// TIA Portal project "Es03_SCHELETRO" (V18)

(* hardware
DEVICE "S71500/ET200MP station_1"  S7-1500 station
   slot 0: "Telaio di montaggio_0"  Rack  6ES7 590-1***0-0AA0
   slot 1: "PLC_1"  CPU 1516-3 PN/DP  6ES7 516-3AN01-0AB0  V2.5
      slot 3: "Display CPU_1"  6ES7591-1BA00-0AA0
   slot 2: "DI 32x24VDC HF_1"  DI 32x24VDC HF  6ES7 521-1BL00-0AB0  V2.1
   slot 3: "DQ 32x24VDC/0.5A HF_1"  DQ 32x24VDC/0.5A HF  6ES7 522-1BL01-0AB0  V1.0
   slot 4: "AI 8xU/I/RTD/TC ST_1"  AI 8xU/I/RTD/TC ST  6ES7 531-7KF00-0AB0  V2.1
   slot 5: "AQ 4xU/I ST_1"  AQ 4xU/I ST  6ES7 532-5HD00-0AB0  V2.1
*)

// ===== PLC "PLC_1"  CPU 1516-3 PN/DP =====

DATA_BLOCK "DB_Comandi"   // DB1
{ S7_Optimized_Access := 'TRUE' }
VERSION : 0.1
   VAR
      btnStop : Bool;
      btnAuto : Bool;
      btnMan : Bool;
      btnReset : Bool;
      btnEmergenza : Bool;
   END_VAR
BEGIN
END_DATA_BLOCK

DATA_BLOCK "DB_Stati"   // DB2
{ S7_Optimized_Access := 'TRUE' }
VERSION : 0.1
   VAR
      sAuto : Bool;
      sStop : Bool;
      sMan : Bool;
      sHome : Bool;
      sAttesaStop : Bool;
      sEmergenza : Bool;
      blni1 : Bool;
      blni2 : Bool;
      bRip1 : Bool;
      bRip2 : Bool;
   END_VAR
BEGIN
END_DATA_BLOCK

DATA_BLOCK "DB_Tappe"   // DB3
{ S7_Optimized_Access := 'TRUE' }
VERSION : 0.1
   VAR
      tappeGemma : Int;
      tappeM1 : Int;
      tappeM2 : Int;
   END_VAR
BEGIN
END_DATA_BLOCK

DATA_BLOCK "DB_Variabili"   // DB4
{ S7_Optimized_Access := 'TRUE' }
VERSION : 0.1
   VAR
      timerResetPulsantiSTART : Bool;
      timerResetPulsantiDONE : Bool;
      timerResetPulsantiOUTPUT : Time;
      timerResetPulsantiDURATA : Time;
   END_VAR
BEGIN
END_DATA_BLOCK

// folder: System blocks/Program resources

DATA_BLOCK "timerResetPulsanti"   // DB5
{ S7_Optimized_Access := 'TRUE' }
AUTHOR : Simatic
FAMILY : IEC
NAME : IEC_TMR
VERSION : 1.0
// stored: InstanceOfName IEC_TIMER
"IEC_TIMER"
BEGIN
END_DATA_BLOCK

// folder: (top level)

FUNCTION "FC_Gemma" : Void   // FC1, SCL
{ S7_Optimized_Access := 'TRUE' }
VERSION : 0.1
BEGIN
   CASE "DB_Tappe".tappeGemma OF
       0: //Stato di Riposo
           "DB_Stati".sStop := TRUE;
           IF "DB_Comandi".btnAuto = TRUE THEN
               "DB_Tappe".tappeGemma := 1; //Home
               "DB_Stati".sAttesaStop := FALSE;
               "DB_Stati".sAuto := FALSE;
               "DB_Stati".sHome := TRUE;
               "DB_Stati".sMan := FALSE;
               "DB_Stati".sStop := FALSE;
               "DB_Stati".sEmergenza := FALSE;
           ELSE
               IF "DB_Comandi".btnMan = TRUE THEN
                   "DB_Tappe".tappeGemma := 4; //Manuale
                   "DB_Stati".sAttesaStop := FALSE;
                   "DB_Stati".sAuto := FALSE;
                   "DB_Stati".sHome := FALSE;
                   "DB_Stati".sMan := TRUE;
                   "DB_Stati".sStop := FALSE;
                   "DB_Stati".sEmergenza := FALSE;
               END_IF;
           END_IF;

        1: //Stato di Home
            IF "DB_Stati".blni1 = TRUE AND "DB_Stati".blni2 = TRUE THEN
                "DB_Tappe".tappeGemma := 2; //Automatico
                "DB_Stati".sAttesaStop := FALSE;
                "DB_Stati".sAuto := TRUE;
                "DB_Stati".sHome := FALSE;
                "DB_Stati".sMan := FALSE;
                "DB_Stati".sStop := FALSE;
                "DB_Stati".sEmergenza := FALSE;
            END_IF;

        2: //Stato di Automatico
            IF "DB_Comandi".btnStop = TRUE THEN
                "DB_Tappe".tappeGemma := 3; //Attesa Stop
                "DB_Stati".sAttesaStop := TRUE;
                "DB_Stati".sAuto := FALSE;
                "DB_Stati".sHome := FALSE;
                "DB_Stati".sMan := FALSE;
                "DB_Stati".sStop := FALSE;
                "DB_Stati".sEmergenza := FALSE;
            END_IF;

        3: //Stato di Attesa Stop
            IF "DB_Stati".bRip1 = TRUE AND "DB_Stati".bRip2 = TRUE THEN
                "DB_Tappe".tappeGemma := 0; //Stop
                "DB_Stati".sAttesaStop := FALSE;
                "DB_Stati".sAuto := FALSE;
                "DB_Stati".sHome := FALSE;
                "DB_Stati".sMan := FALSE;
                "DB_Stati".sStop := TRUE;
                "DB_Stati".sEmergenza := FALSE;
            END_IF;

        4: //Stato di Manuale
            IF "DB_Comandi".btnStop = TRUE THEN
                "DB_Tappe".tappeGemma := 0; //Stop
                "DB_Stati".sAttesaStop := FALSE;
                "DB_Stati".sAuto := FALSE;
                "DB_Stati".sHome := FALSE;
                "DB_Stati".sMan := FALSE;
                "DB_Stati".sStop := TRUE;
                "DB_Stati".sEmergenza := FALSE;
            END_IF;

        5: //Stato di Emergenza
            IF "DB_Comandi".btnEmergenza = TRUE AND "DB_Stati".sEmergenza THEN
                "DB_Tappe".tappeGemma := 0; //Stop
                "DB_Stati".sAttesaStop := FALSE;
                "DB_Stati".sAuto := FALSE;
                "DB_Stati".sHome := FALSE;
                "DB_Stati".sMan := FALSE;
                "DB_Stati".sStop := TRUE;
                "DB_Stati".sEmergenza := FALSE;
            END_IF;
    END_CASE;

    //Gestione Emergenza
    //
    IF "DB_Comandi".btnEmergenza = FALSE THEN
        "DB_Tappe".tappeGemma := 5; //Emergenza
        "DB_Stati".sAttesaStop := FALSE;
        "DB_Stati".sAuto := FALSE;
        "DB_Stati".sHome := FALSE;
        "DB_Stati".sMan := FALSE;
        "DB_Stati".sStop := FALSE;
        "DB_Stati".sEmergenza := TRUE;
    END_IF;
END_FUNCTION

FUNCTION "FC_Grafset" : Void   // FC2, SCL
{ S7_Optimized_Access := 'TRUE' }
VERSION : 0.1
BEGIN
   //Imposto bIni e bRip a TRUE. Andranno poi gestiti in base alle condizioni dell'impianto
   //
   "DB_Stati".blni1 := TRUE;
   "DB_Stati".blni2 := TRUE;
   "DB_Stati".bRip1 := TRUE;
   "DB_Stati".bRip2 := TRUE;
END_FUNCTION

FUNCTION "FC_ResetPulsanti" : Void   // FC3, SCL
{ S7_Optimized_Access := 'TRUE' }
VERSION : 0.1
BEGIN
   IF "DB_Comandi".btnAuto = TRUE OR
       "DB_Comandi".btnMan = TRUE OR
       "DB_Comandi".btnReset = TRUE OR
       "DB_Comandi".btnStop = TRUE THEN
       "DB_Variabili".timerResetPulsantiSTART := TRUE;
   END_IF;

   IF "DB_Variabili".timerResetPulsantiDONE = TRUE THEN
       "DB_Variabili".timerResetPulsantiSTART := FALSE;
       "DB_Variabili".timerResetPulsantiDONE := FALSE;
       "DB_Comandi".btnAuto := FALSE;
       "DB_Comandi".btnMan := FALSE;
       "DB_Comandi".btnReset := FALSE;
       "DB_Comandi".btnStop := FALSE;
   END_IF;
END_FUNCTION

FUNCTION "FC_Timer" : Void   // FC4, SCL
{ S7_Optimized_Access := 'TRUE' }
VERSION : 0.1
BEGIN
   "DB_Variabili".timerResetPulsantiDURATA := T#500ms;

   "timerResetPulsanti".TON(IN:="DB_Variabili".timerResetPulsantiSTART,
                            PT:="DB_Variabili".timerResetPulsantiDURATA,
                            Q=>"DB_Variabili".timerResetPulsantiDONE,
                            ET=>"DB_Variabili".timerResetPulsantiOUTPUT);
END_FUNCTION

FUNCTION "FC_Uscite" : Void   // FC5, SCL
{ S7_Optimized_Access := 'TRUE' }
VERSION : 0.1
BEGIN
END_FUNCTION

ORGANIZATION_BLOCK "Main"   // OB1, LAD, ProgramCycle
TITLE = "Main Program Sweep (Cycle)"
{ S7_Optimized_Access := 'TRUE' }
VERSION : 0.1
   VAR_INPUT
      Initial_Call : Bool;   // Initial call of this OB
      Remanence : Bool;   // =True, if remanent data are available
   END_VAR
   VAR_TEMP   // added for the SCL form of the ladder/FBD networks
      _w1 : Bool;
      _w2 : Bool;
      _w3 : Bool;
      _w4 : Bool;
   END_VAR
BEGIN

REGION Network 1
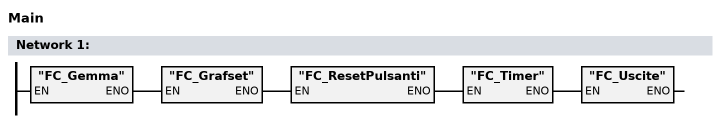
   RUNG wire#powerrail
      "FC_Gemma"()
      "FC_Grafset"()
      "FC_ResetPulsanti"()
      "FC_Timer"()
      "FC_Uscite"()
   END_RUNG
   // the same network as SCL:
   "FC_Gemma"(ENO => #_w1);
   "FC_Grafset"(EN := #_w1, ENO => #_w2);
   "FC_ResetPulsanti"(EN := #_w2, ENO => #_w3);
   "FC_Timer"(EN := #_w3, ENO => #_w4);
   IF #_w4 THEN "FC_Uscite"(); END_IF;
END_REGION
END_ORGANIZATION_BLOCK